// TIA Portal V20 export
TYPE "typeCmControlNodeInterlock"
// stored: Namespace Unit1.Em2
   STRUCT
      ElectrodeFixRightTop { ExternalWritable := 'False'} : "LER_typeTwoWayActuatorInterlock";
      ElectrodeFixRightBottom { ExternalWritable := 'False'} : "LER_typeTwoWayActuatorInterlock";
      ElectrodeFixLeftTopX { ExternalWritable := 'False'} : "LER_typeTwoWayActuatorInterlock";
      ElectrodeFixLeftBottomX { ExternalWritable := 'False'} : "LER_typeTwoWayActuatorInterlock";
      ElectrodeFixLeftTopZ { ExternalWritable := 'False'} : "LER_typeTwoWayActuatorInterlock";
      ElectrodeFixLeftBottomZ { ExternalWritable := 'False'} : "LER_typeTwoWayActuatorInterlock";
      UwSemiSplicerVacuumRightTop { ExternalWritable := 'False'} : "LER_typeTwoWayActuatorInterlock";
      UwSemiSplicerVacuumRightBottom { ExternalWritable := 'False'} : "LER_typeTwoWayActuatorInterlock";
      UwSemiSplicerVacuumLeftTop { ExternalWritable := 'False'} : "LER_typeTwoWayActuatorInterlock";
      UwSemiSplicerVacuumLeftBottom { ExternalWritable := 'False'} : "LER_typeTwoWayActuatorInterlock";
      ElectrodeCutter { ExternalWritable := 'False'} : "LER_typeTwoWayActuatorInterlock";
      SplicingLeftModuleMover { ExternalWritable := 'False'} : "LER_typeTwoWayActuatorInterlock";
      SplicingRightModuleMover { ExternalWritable := 'False'} : "LER_typeTwoWayActuatorInterlock";
      ElectrodeLeftHolderMover { ExternalWritable := 'False'} : "LER_typeTwoWayActuatorInterlock";
      ElectrodeRightHolderMover { ExternalWritable := 'False'} : "LER_typeTwoWayActuatorInterlock";
      TapeLoadingTurn { ExternalWritable := 'False'} : "LER_typeTwoWayActuatorInterlock";
      TapeAttachUnit { ExternalWritable := 'False'} : "LER_typeTwoWayActuatorInterlock";
      UWSemiSplicerTapeVacuum { ExternalWritable := 'False'} : "LER_typeTwoWayActuatorInterlock";
      Stopper { ExternalWritable := 'False'} : "LER_typeTwoWayActuatorInterlock";
      SupportUnitTransfer { ExternalWritable := 'False'} : "LER_typeTwoWayActuatorInterlock";
      SupportUnitShaft { ExternalWritable := 'False'} : "LER_typeTwoWayActuatorInterlock";
      FrameCover { ExternalWritable := 'False'} : "LER_typeTwoWayActuatorInterlock";
   END_STRUCT;
END_TYPE
